// TIA Portal V18 export
// export: Created 2026-06-11T12:00:00Z, ExportSetting WithDefaults
AlarmLogging "AlarmLogging_1"
  AnalogAlarm "AI_Alarm_TT32_HiHi"  DelayTimeUnit=Seconds, LimitMode=HighHigh, LimitValue=78, Priority=3, AlarmText="<body><p>CẢNH BÁO NGUY HIỂM: Nhiệt độ TT32 quá cao! Giá trị = {0} °C (Ngưỡng: 78°C)</p></body>"
    AlarmClass   AlarmClass=Errors
    AnalogAlarmTag   Tag=1400_TT32_PV
  AnalogAlarm "AI_Alarm_TT32_Hi"  DelayTimeUnit=Seconds, LimitMode=High, LimitValue=75, Priority=2, AlarmText="<body><p>CẢNH BÁO: Nhiệt độ TT32 cao! Giá trị = {0} °C (Ngưỡng: 75°C)</p></body>"
    AlarmClass   AlarmClass=Errors
    AnalogAlarmTag   Tag=1400_TT32_PV
  AnalogAlarm "AI_Alarm_TX35_HiHi"  DelayTimeUnit=Seconds, LimitMode=HighHigh, LimitValue=8.0, Priority=3, AlarmText="<body><p>CẢNH BÁO NGUY HIỂM: Áp suất TX35 quá cao! Giá trị = {0} bar (Ngưỡng: 8 bar)</p></body>"
    AlarmClass   AlarmClass=Errors
    AnalogAlarmTag   Tag=1406_TX35_PV
  AnalogAlarm "AI_Alarm_TX35_Hi"  DelayTimeUnit=Seconds, LimitMode=High, LimitValue=7.0, Priority=2, AlarmText="<body><p>CẢNH BÁO: Áp suất TX35 cao! Giá trị = {0} bar (Ngưỡng: 7 bar)</p></body>"
    AlarmClass   AlarmClass=Errors
    AnalogAlarmTag   Tag=1406_TX35_PV
